FUNCTION_BLOCK FB_NoNet
VAR_INPUT
END_VAR
VAR_OUTPUT
END_VAR
VAR
END_VAR

END_FUNCTION_BLOCK

(* stored: Version 1.1.0.1, ProductVersion 3.1.0.36
   POU FB_NoNet: Id {31b9d237-ce64-4f6d-b9e1-c64e2c4e62d4}, SpecialFunc None *)
